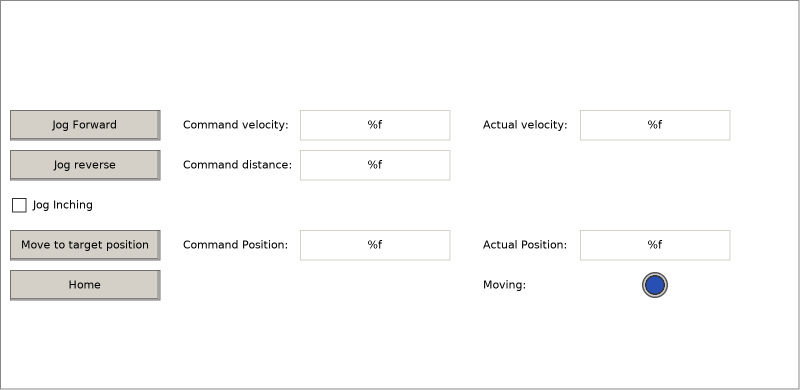
VISUALIZATION VisuAxisControl  // 800x390
    Button (10,110 150x30), "Jog Forward"
        tap GVL_DevManual.fbManualControler.pDevAxis^.stManualCtrl.bCmdJogForward
    Button (10,150 150x30), "Jog reverse"
        tap GVL_DevManual.fbManualControler.pDevAxis^.stManualCtrl.bCmdJogReverse
    Button (10,230 150x30), "Move to target position"
        tap GVL_DevManual.fbManualControler.pDevAxis^.stManualCtrl.bCmdToPos
    Button (10,270 150x30), "Home"
        tap GVL_DevManual.fbManualControler.pDevAxis^.stManualCtrl.bCmdHome
    Checkbox (10,190 150x30), "Jog Inching", variable: GVL_DevManual.fbManualControler.pDevAxis^.stManualCtrl.bCmdInching
    Label (180,150 120x30), "Command distance:"
    Label (180,110 120x30), "Command velocity:"
    Label (180,230 120x30), "Command Position:"
    Textfield (300,110 150x30), "%f", text variable: GVL_DevManual.fbManualControler.pDevAxis^.stManualCtrl.fVelocity
        OnMouseDown: write the text variable via VisuDialogs.Numpad
    Textfield (300,150 150x30), "%f", text variable: GVL_DevManual.fbManualControler.pDevAxis^.stManualCtrl.fDistance
        OnMouseDown: write the text variable via VisuDialogs.Numpad
    Textfield (300,230 150x30), "%f", text variable: GVL_DevManual.fbManualControler.pDevAxis^.stManualCtrl.fPosition
        OnMouseDown: write the text variable via VisuDialogs.Numpad
    Label (480,110 100x30), "Actual velocity:"
    Label (480,230 100x30), "Actual Position:"
    Textfield (580,230 150x30), "%f", text variable: GVL_DevManual.fbManualControler.pDevAxis^.fActPosition
        OnMouseDown: write the text variable via VisuDialogs.Numpad
    Textfield (580,110 150x30), "%f", text variable: GVL_DevManual.fbManualControler.pDevAxis^.fVelocity
        OnMouseDown: write the text variable via VisuDialogs.Numpad
    Lamp1 (580,270 150x30), variable: GVL_DevManual.fbManualControler.pDevAxis^.AxisRef.Status.Moving, style: Lamp-Lamp1-Blue
    Label (480,270 100x30), "Moving:"
END_VISUALIZATION

(* stored: Version 1.1.0.1, ProductVersion 3.1.4024.5
   Visu VisuAxisControl: Id {3f99e6a2-4ef1-4500-aca5-d6ca766f4789} *)
